PROGRAM MAIN
VAR
	sFilePathName	: STRING := 'C:\TwinCAT\CNC\TestNci1.txt';
	sErrorMessage	: STRING := '';
	bOpen			: BOOL;
	bClose 			: BOOL;
	bSave 			: BOOL;
	bNew			: BOOL;
	nErrorCode		: USINT;
	nLineNumber		: USINT;
	bEnable: BOOL;
END_VAR

(*V03 	- 28.09.2017 13:40*)
(*V03.1 - 10.02.2017 *)

sErrorMessage	:= VisuFctTextEditorGetErrorText(usiErrCode := nErrorCode);

PRG_NcControl();
//PRG_MFuncControl();
PRG_Kinematic();

//PRG_Process();

//PRG_OpcUA();


IF bEnable THEN
	stAxisM1_B.In.xEnable	:= TRUE;
	stAxisM2_C.In.xEnable	:= TRUE;
	stAxisM3_A.In.xEnable	:= TRUE;
	stAxisX.In.xEnable	:= TRUE;
	stAxisY.In.xEnable	:= TRUE;
	stAxisZ.In.xEnable	:= TRUE;
	
	stAxisM1_B.In.fOverride	:= 100;
	stAxisM2_C.In.fOverride	:= 100;
	stAxisM3_A.In.fOverride	:= 100;
	stAxisX.In.fOverride	:= 100;
	stAxisY.In.fOverride	:= 100;
	stAxisZ.In.fOverride	:= 100;
ELSE
	stAxisM1_B.In.xEnable	:= FALSE;
	stAxisM2_C.In.xEnable	:= FALSE;
	stAxisM3_A.In.xEnable	:= FALSE;
	stAxisX.In.xEnable	:= FALSE;
	stAxisY.In.xEnable	:= FALSE;
	stAxisZ.In.xEnable	:= FALSE;
END_IF

stAxisX.In.fSetPos;
stAxisY.In.fSetPos;
stAxisZ.In.fSetPos;

stAxisX.In.fSetVelo;
stAxisY.In.fSetVelo;
stAxisZ.In.fSetVelo;

stAxisX.In.xMove;
stAxisY.In.xMove;
stAxisZ.In.xMove;


AxisM1PosValue	:= AxisM1_B.NcToPlc.ActPos;
AxisM2PosValue	:= AxisM2_C.NcToPlc.ActPos;
AxisM3PosValue	:= AxisM3_A.NcToPlc.ActPos;

AxisM1VeloValue	:= AxisM1_B.NcToPlc.ActVelo;
AxisM2VeloValue	:= AxisM2_C.NcToPlc.ActVelo;
AxisM3VeloValue	:= AxisM3_A.NcToPlc.ActVelo;

END_PROGRAM

(* stored: Version 1.1.0.1, ProductVersion 3.1.4024.0
   POU MAIN: Id {2020bd6b-90a0-4fc7-9a1c-76bd8c902114}, SpecialFunc None *)
